FUNCTION_BLOCK DecodeINeredaAct (* Composite Function Block Type *)
  (* Standard: 61499-2 *)
  (* Version 0.0, 6/7/2026, Schneider Electric, template *)
  PACKAGE SE.Nereda;
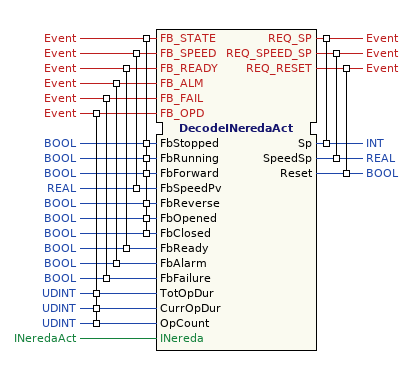
  EVENT_INPUT
    FB_STATE WITH FbStopped, FbRunning, FbForward, FbReverse, FbOpened, FbClosed;
    FB_SPEED WITH FbSpeedPv;
    FB_READY WITH FbReady;
    FB_ALM WITH FbAlarm;
    FB_FAIL WITH FbFailure;
    FB_OPD WITH TotOpDur, CurrOpDur, OpCount;
  END_EVENT
  EVENT_OUTPUT
    REQ_SP WITH Sp;
    REQ_SPEED_SP WITH SpeedSp;
    REQ_RESET WITH Reset;
  END_EVENT
  VAR_INPUT
    FbStopped : BOOL;
    FbRunning : BOOL;
    FbForward : BOOL;
    FbSpeedPv : REAL;
    FbReverse : BOOL;
    FbOpened : BOOL;
    FbClosed : BOOL;
    FbReady : BOOL;
    FbAlarm : BOOL;
    FbFailure : BOOL;
    TotOpDur : UDINT;
    CurrOpDur : UDINT;
    OpCount : UDINT;
  END_VAR
  VAR_OUTPUT
    Sp : INT;
    SpeedSp : REAL;
    Reset : BOOL;
  END_VAR
  SOCKETS
    INereda : INeredaAct;
  END_SOCKETS
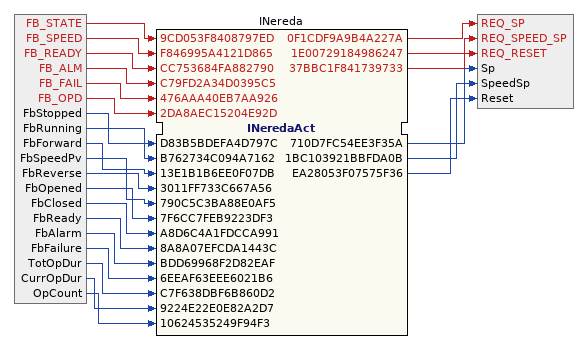
  EVENT_CONNECTIONS
    FB_STATE TO INereda.9CD053F8408797ED;
    FB_SPEED TO INereda.F846995A4121D865;
    FB_READY TO INereda.CC753684FA882790;
    FB_ALM TO INereda.C79FD2A34D0395C5;
    FB_FAIL TO INereda.476AAA40EB7AA926;
    FB_OPD TO INereda.2DA8AEC15204E92D;
    INereda.0F1CDF9A9B4A227A TO REQ_SP;
    INereda.1E00729184986247 TO REQ_SPEED_SP;
    INereda.37BBC1F841739733 TO REQ_RESET;
  END_CONNECTIONS
  DATA_CONNECTIONS
    FbStopped TO INereda.D83B5BDEFA4D797C;
    FbRunning TO INereda.B762734C094A7162;
    FbForward TO INereda.13E1B1B6EE0F07DB;
    FbReverse TO INereda.3011FF733C667A56;
    FbSpeedPv TO INereda.790C5C3BA88E0AF5;
    FbOpened TO INereda.7F6CC7FEB9223DF3;
    FbClosed TO INereda.A8D6C4A1FDCCA991;
    FbReady TO INereda.8A8A07EFCDA1443C;
    FbAlarm TO INereda.BDD69968F2D82EAF;
    FbFailure TO INereda.6EEAF63EEE6021B6;
    TotOpDur TO INereda.C7F638DBF6B860D2;
    CurrOpDur TO INereda.9224E22E0E82A2D7;
    OpCount TO INereda.10624535249F94F3;
    INereda.710D7FC54EE3F35A TO Sp;
    INereda.1BC103921BBFDA0B TO SpeedSp;
    INereda.EA28053F07575F36 TO Reset;
  END_CONNECTIONS
END_FUNCTION_BLOCK
